// TIA Portal V19 export
FUNCTION_BLOCK "F_Zone20_FB"   // FB188, F_LAD
TITLE = SAFETY ZONE 11 - AREA 02 (PROFILATRICE)
// -
// stored: Access Published
   VAR
      FNS : "ForceNormalStop";
      F_Sinamics_Rollformer : "FDevice_Sinamics_FB";
   END_VAR
   VAR_TEMP
      DoorNormalStop : Bool;
      DoorSafeStop : Bool;
      Door_Ok : Bool;
   END_VAR
   VAR CONSTANT
      ROLLFORMER_S120_STOPPING_TIME : Time := T#1S;
   END_VAR
BEGIN

REGION Network 1: < < < < < < < < < < DOOR > > > > > > > > > >
END_REGION

REGION Network 2: Zone Entry enable
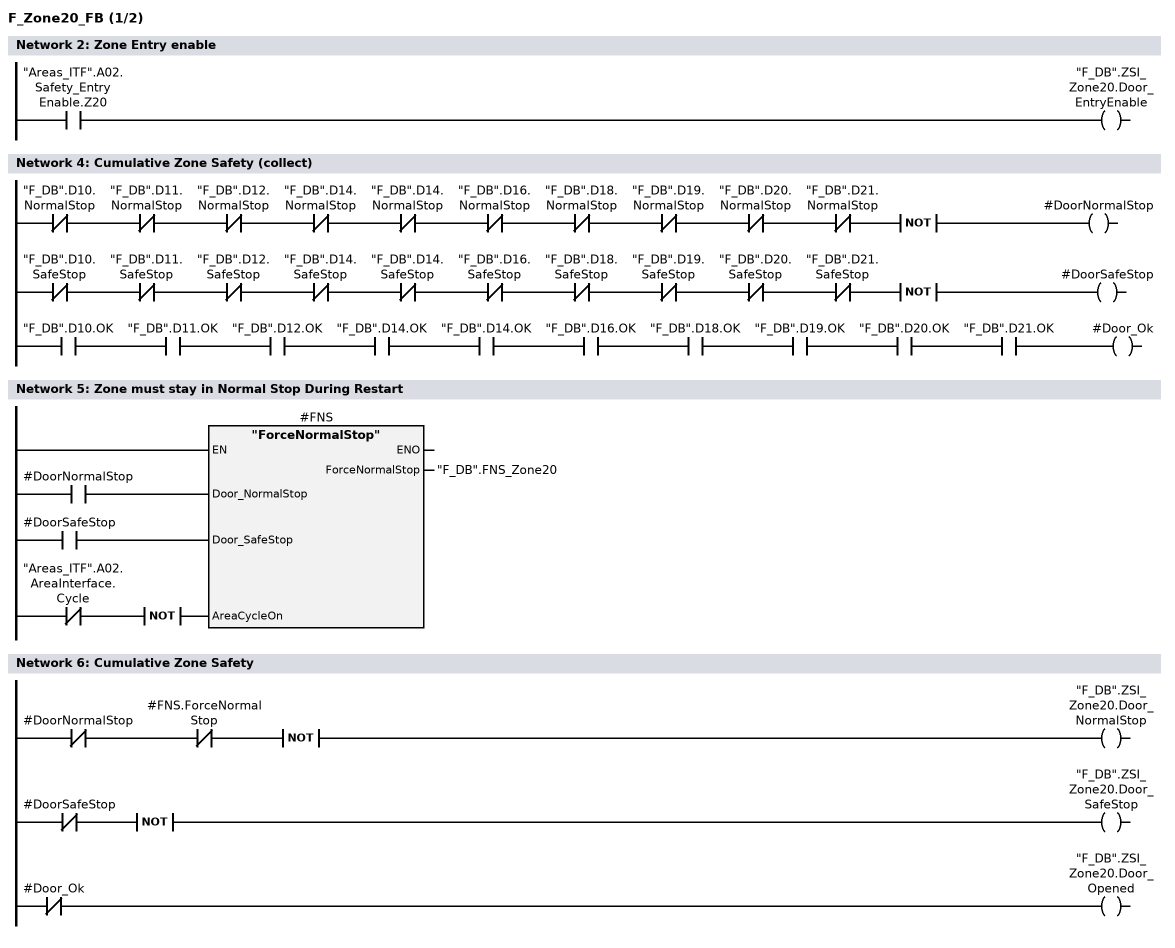
   RUNG wire#powerrail
      Contact( "Areas_ITF".A02.Safety_EntryEnable.Z20 )
      Coil( "F_DB".ZSI_Zone20.Door_EntryEnable )
   END_RUNG
   // the same network as SCL:
   "F_DB".ZSI_Zone20.Door_EntryEnable := "Areas_ITF".A02.Safety_EntryEnable.Z20;
END_REGION

REGION Network 3: < < < < < < < < < < ZONE SAFETY INTERFACE > > > > > > > > > >
END_REGION

REGION Network 4: Cumulative Zone Safety (collect)
   RUNG wire#powerrail
      I_Contact( "F_DB".D10.NormalStop )
      I_Contact( "F_DB".D11.NormalStop )
      I_Contact( "F_DB".D12.NormalStop )
      I_Contact( "F_DB".D14.NormalStop )
      I_Contact( "F_DB".D14.NormalStop )
      I_Contact( "F_DB".D16.NormalStop )
      I_Contact( "F_DB".D18.NormalStop )
      I_Contact( "F_DB".D19.NormalStop )
      I_Contact( "F_DB".D20.NormalStop )
      I_Contact( "F_DB".D21.NormalStop )
      Not()
      Coil( #DoorNormalStop )
   END_RUNG
   RUNG wire#powerrail
      I_Contact( "F_DB".D10.SafeStop )
      I_Contact( "F_DB".D11.SafeStop )
      I_Contact( "F_DB".D12.SafeStop )
      I_Contact( "F_DB".D14.SafeStop )
      I_Contact( "F_DB".D14.SafeStop )
      I_Contact( "F_DB".D16.SafeStop )
      I_Contact( "F_DB".D18.SafeStop )
      I_Contact( "F_DB".D19.SafeStop )
      I_Contact( "F_DB".D20.SafeStop )
      I_Contact( "F_DB".D21.SafeStop )
      Not()
      Coil( #DoorSafeStop )
   END_RUNG
   RUNG wire#powerrail
      Contact( "F_DB".D10.OK )
      Contact( "F_DB".D11.OK )
      Contact( "F_DB".D12.OK )
      Contact( "F_DB".D14.OK )
      Contact( "F_DB".D14.OK )
      Contact( "F_DB".D16.OK )
      Contact( "F_DB".D18.OK )
      Contact( "F_DB".D19.OK )
      Contact( "F_DB".D20.OK )
      Contact( "F_DB".D21.OK )
      Coil( #Door_Ok )
   END_RUNG
   // the same network as SCL:
   #DoorNormalStop := NOT (NOT "F_DB".D10.NormalStop AND NOT "F_DB".D11.NormalStop AND NOT "F_DB".D12.NormalStop AND NOT "F_DB".D14.NormalStop AND NOT "F_DB".D14.NormalStop AND NOT "F_DB".D16.NormalStop AND NOT "F_DB".D18.NormalStop AND NOT "F_DB".D19.NormalStop AND NOT "F_DB".D20.NormalStop AND NOT "F_DB".D21.NormalStop);
   #DoorSafeStop := NOT (NOT "F_DB".D10.SafeStop AND NOT "F_DB".D11.SafeStop AND NOT "F_DB".D12.SafeStop AND NOT "F_DB".D14.SafeStop AND NOT "F_DB".D14.SafeStop AND NOT "F_DB".D16.SafeStop AND NOT "F_DB".D18.SafeStop AND NOT "F_DB".D19.SafeStop AND NOT "F_DB".D20.SafeStop AND NOT "F_DB".D21.SafeStop);
   #Door_Ok := "F_DB".D10.OK AND "F_DB".D11.OK AND "F_DB".D12.OK AND "F_DB".D14.OK AND "F_DB".D14.OK AND "F_DB".D16.OK AND "F_DB".D18.OK AND "F_DB".D19.OK AND "F_DB".D20.OK AND "F_DB".D21.OK;
END_REGION

REGION Network 5: Zone must stay in Normal Stop During Restart
   RUNG wire#powerrail
      #FNS(Door_NormalStop := wire#w1, Door_SafeStop := wire#w2, AreaCycleOn := wire#w3, ForceNormalStop => "F_DB".FNS_Zone20)
   END_RUNG
   RUNG wire#powerrail
      Contact( #DoorNormalStop )
   END_RUNG wire#w1
   RUNG wire#powerrail
      Contact( #DoorSafeStop )
   END_RUNG wire#w2
   RUNG wire#powerrail
      I_Contact( "Areas_ITF".A02.AreaInterface.Cycle )
      Not()
   END_RUNG wire#w3
   // the same network as SCL:
   #FNS(Door_NormalStop := #DoorNormalStop,   // "ForceNormalStop"
        Door_SafeStop := #DoorSafeStop,
        AreaCycleOn := NOT (NOT "Areas_ITF".A02.AreaInterface.Cycle),
        ForceNormalStop => "F_DB".FNS_Zone20);
END_REGION

REGION Network 6: Cumulative Zone Safety
   RUNG wire#powerrail
      I_Contact( #DoorNormalStop )
      I_Contact( #FNS.ForceNormalStop )
      Not()
      Coil( "F_DB".ZSI_Zone20.Door_NormalStop )
   END_RUNG
   RUNG wire#powerrail
      I_Contact( #DoorSafeStop )
      Not()
      Coil( "F_DB".ZSI_Zone20.Door_SafeStop )
   END_RUNG
   RUNG wire#powerrail
      I_Contact( #Door_Ok )
      Coil( "F_DB".ZSI_Zone20.Door_Opened )
   END_RUNG
   // the same network as SCL:
   "F_DB".ZSI_Zone20.Door_NormalStop := NOT (NOT #DoorNormalStop AND NOT #FNS.ForceNormalStop);
   "F_DB".ZSI_Zone20.Door_SafeStop := NOT (NOT #DoorSafeStop);
   "F_DB".ZSI_Zone20.Door_Opened := NOT #Door_Ok;
END_REGION

REGION Network 7: >
END_REGION

REGION Network 8: >
END_REGION

REGION Network 9: < < < < < < < < < < DEVICES SAFETY VALVES > > > > > > > > > >
END_REGION

REGION Network 10: >
END_REGION

REGION Network 11: >
END_REGION

REGION Network 12: < < < < < < < < < < DEVICES CONTACTORS > > > > > > > > > >
END_REGION

REGION Network 13: >
END_REGION

REGION Network 14: >
END_REGION

REGION Network 15: < < < < < < < < < < DEVICES S120 > > > > > > > > > >
END_REGION

REGION Network 16: S120 - Rollformer
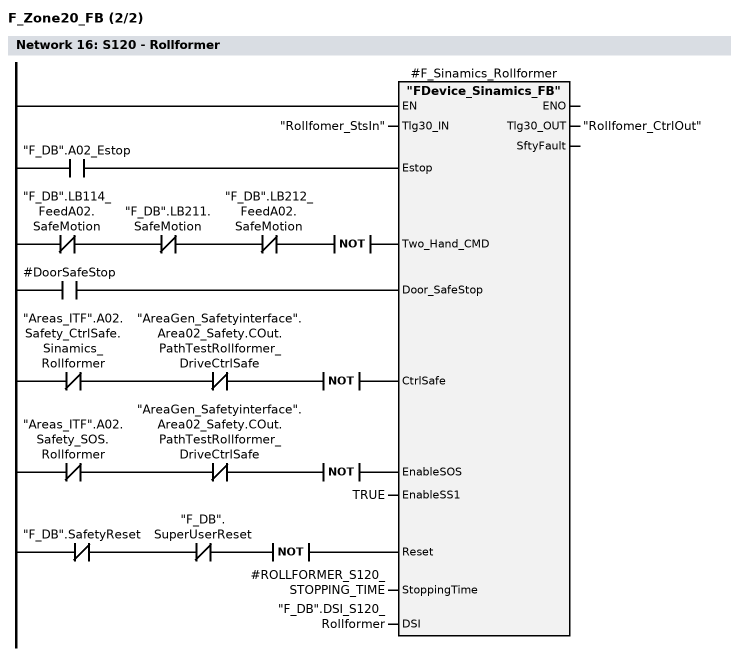
   RUNG wire#powerrail
      #F_Sinamics_Rollformer(Estop := wire#w1, Two_Hand_CMD := wire#w2, Door_SafeStop := wire#w3, CtrlSafe := wire#w4, EnableSOS := wire#w5, Reset := wire#w6, Tlg30_IN := "Rollfomer_StsIn", EnableSS1 := TRUE, StoppingTime := #ROLLFORMER_S120_STOPPING_TIME, DSI := "F_DB".DSI_S120_Rollformer, Tlg30_OUT => "Rollfomer_CtrlOut", SftyFault =>)
   END_RUNG
   RUNG wire#powerrail
      Contact( "F_DB".A02_Estop )
   END_RUNG wire#w1
   RUNG wire#powerrail
      I_Contact( "F_DB".LB114_FeedA02.SafeMotion )
      I_Contact( "F_DB".LB211.SafeMotion )
      I_Contact( "F_DB".LB212_FeedA02.SafeMotion )
      Not()
   END_RUNG wire#w2
   RUNG wire#powerrail
      Contact( #DoorSafeStop )
   END_RUNG wire#w3
   RUNG wire#powerrail
      I_Contact( "Areas_ITF".A02.Safety_CtrlSafe.Sinamics_Rollformer )
      I_Contact( "AreaGen_Safetyinterface".Area02_Safety.COut.PathTestRollformer_DriveCtrlSafe )
      Not()
   END_RUNG wire#w4
   RUNG wire#powerrail
      I_Contact( "Areas_ITF".A02.Safety_SOS.Rollformer )
      I_Contact( "AreaGen_Safetyinterface".Area02_Safety.COut.PathTestRollformer_DriveCtrlSafe )
      Not()
   END_RUNG wire#w5
   RUNG wire#powerrail
      I_Contact( "F_DB".SafetyReset )
      I_Contact( "F_DB".SuperUserReset )
      Not()
   END_RUNG wire#w6
   // the same network as SCL:
   #F_Sinamics_Rollformer(Tlg30_IN := "Rollfomer_StsIn",   // "FDevice_Sinamics_FB"
                          Estop := "F_DB".A02_Estop,
                          Two_Hand_CMD := NOT (NOT "F_DB".LB114_FeedA02.SafeMotion AND NOT "F_DB".LB211.SafeMotion AND NOT "F_DB".LB212_FeedA02.SafeMotion),
                          Door_SafeStop := #DoorSafeStop,
                          CtrlSafe := NOT (NOT "Areas_ITF".A02.Safety_CtrlSafe.Sinamics_Rollformer AND NOT "AreaGen_Safetyinterface".Area02_Safety.COut.PathTestRollformer_DriveCtrlSafe),
                          EnableSOS := NOT (NOT "Areas_ITF".A02.Safety_SOS.Rollformer AND NOT "AreaGen_Safetyinterface".Area02_Safety.COut.PathTestRollformer_DriveCtrlSafe),
                          EnableSS1 := TRUE,
                          Reset := NOT (NOT "F_DB".SafetyReset AND NOT "F_DB".SuperUserReset),
                          StoppingTime := #ROLLFORMER_S120_STOPPING_TIME,
                          DSI := "F_DB".DSI_S120_Rollformer,
                          Tlg30_OUT => "Rollfomer_CtrlOut");
END_REGION

REGION Network 17: >
END_REGION

REGION Network 18: >
END_REGION
END_FUNCTION_BLOCK
